TYPE ST_ProdPar :
STRUCT
	InMoldDrying			: ST_IMDProdPar;
	ProductHandling			: ST_ProductHandlingProdPar;

END_STRUCT
END_TYPE

(* stored: Version 1.1.0.1, ProductVersion 3.1.4020.12
   DUT ST_ProdPar: Id {f6477087-9b47-4999-8080-aaf6d1beeb4c} *)
